FUNCTION_BLOCK J_Stop_Testing_SM
VAR_INPUT
	JST_NodeID					: BYTE; (* This Port No. addresses the CANopen Node (see System Manager) *)
	JST_Start_Testing			: BOOL; (* Send True to start the Stop Testing*)
	JST_Statusword				: WORD;	
	JST_Current_State 			: E_Statemachine_State;
END_VAR
VAR_OUTPUT
	Finished 				: BOOL;
	JST_Controlword 		: WORD;
	Mode_of_operation 		: E_Mode_of_operation	:= E_Mode_of_operation.No_mode_active;
END_VAR
VAR
	JST_Profile_Velocity_Mode 		: Profile_Velocity_Mode;
	e_Stop_Testing_State_Machine 	: (Idle,
									   Start_Drive, 
									   Check_Start_Drive_Condition,
								       Stop_Testing, 
									   Check_Stop_Drive_Condition,
									   Error_Handling) := Idle; 
									
	e_Operation_Mode : E_Mode_of_operation := E_Mode_of_operation.Profile_position_mode;
	
	e_Stop_Mode :  (Switch_On,					//schnell runterrampen -> Switched on
					Shutdown,					//Disable PS
					Disable_Voltage,			//Disable PS
					Vel_To_Zero,				//Ramp down
					Halt,						//stillstand mit dehmoment -> Weiterdrehen
					Quick_Stop,					//schnell runterrampen -> Switch on Disabled
					Fault,						//DISABLE PS
					STO1,						//Disable PS
					STO2,						//Disable PS
					END) := Switch_On;
					
	e_Stop_Type :  (Idle_Output_Stage,
				    Ramp_Down,
					Vel_Zero,
					Quick_Stop);
					
	
	JST_Profile_velocity_parameters	: ST_Velocity_parameters := (vl_target_velocity 	  := 1000,
																 vl_velocity_acceleration := 1000,
																 vl_velocity_deceleration := 1000);
	vl_target_velocity	: INT := 0;
	Target_State: E_STATEMACHINE_STATE;
	
	SDO_WRITE		: FB_SDO_WRITE;
	WriteData		: ARRAY [0..255] OF BYTE;
	
	Tolerance : INT := 30;		//Assumed that unit is RPM
	
	// Trash Variables 
	Temp : BOOL := TRUE;
	JumpNextState : BOOL := FALSE;
	
END_VAR

CASE e_Stop_Testing_State_Machine OF
	
	Idle:
		IF JST_Start_Testing THEN
			e_Stop_Testing_State_Machine := Start_Drive;
		ELSE
			e_Stop_Testing_State_Machine := Idle;
		END_IF
		
//---------------------Start Drive SM-----------------------------------
	Start_Drive:
	
		CASE e_Operation_Mode OF
			
			e_Operation_Mode.Profile_position_mode:
				// Vel = 1000 ; Acc = 1000 ; Dec = 1000, Pos = 10000000	
				IF NOT JST_Profile_Velocity_Mode.Finished THEN
					//just want to set acc and dec but not enable the drive
					JST_Profile_Velocity_Mode (NodeID := JST_NodeID,		//PVM just because the param for acc and dec are set and the same as in PPM
						   Start := TRUE,
						   Current_State := JST_Current_State,
						   Statusword := JST_Statusword,
						   Profile_velocity_parameters := JST_Profile_velocity_parameters,
						   Controlword => JST_Controlword);
					JST_Controlword := CONTROLWORD_STATE_CHANGE(JST_Current_State, E_Statemachine_State.Switch_on_disabled);
				ELSE
					WHILE Temp = TRUE DO
						PDO.Mode_of_operation 	:= E_Mode_of_operation.Profile_position_mode;		//Maybe its enought to set it once?
						PDO.Profile_velocity := JST_Profile_velocity_parameters.vl_target_velocity;
						Temp := FALSE;
					END_WHILE
					JST_Controlword := CONTROLWORD_STATE_CHANGE(JST_Current_State, E_statemachine_state.Operation_enabled);
					e_Stop_Testing_State_Machine := Check_Start_Drive_Condition;
				END_IF
								
			e_Operation_Mode.Velocity_mode:
				// Vel = 1000
				// // Start Drive, Wait for SDO written then change state
				e_Stop_Testing_State_Machine := Check_Start_Drive_Condition;
				
			e_Operation_Mode.Profile_velocity_mode:
				// Vel = 1000 ; Acc = 1000 ; Dec = 500
				// Start Drive, Wait for SDO written then change state
				e_Stop_Testing_State_Machine := Check_Start_Drive_Condition;
				
			e_Operation_Mode.Profile_torque_mode:
				// Torque = 100 pro mill
				// Start Drive, Wait for SDO written then change state
				e_Stop_Testing_State_Machine := Check_Start_Drive_Condition;
		END_CASE
		
		
//------------------Check Drive Condition SM-----------------------------
	Check_Start_Drive_Condition:
	
		CASE e_Operation_Mode OF
			
			e_Operation_Mode.Profile_position_mode:
				IF ABS(PDO.Velocity_actual_value - JST_Profile_velocity_parameters.vl_target_velocity) < Tolerance THEN
					e_Stop_Testing_State_Machine := Stop_Testing;
				ELSE
					;
				END_IF
				// Wait for desired speed 
				// true change state / false wirte msg log
			e_Operation_Mode.Velocity_mode:
				// Wait for desired speed 
				// true change state / false wirte msg log
			e_Operation_Mode.Profile_velocity_mode:
				// Check acc and dec
				// Wait for desired speed 
				// true change state / false wirte msg log
			e_Operation_Mode.Profile_torque_mode:
				// check torque
				// true change state / false wirte msg log
		END_CASE
		
//------------------Stop Testing SM--------------------------------------		
	Stop_Testing:
	
		CASE e_Operation_Mode OF
		//----------testing in Profile Position Mode---------------------
			e_Operation_Mode.Profile_position_mode:
					
				CASE e_Stop_Mode OF
					Switch_On:
						//Trigger Stopp
						e_Stop_Mode := Shutdown;
						e_Stop_Type := Idle_Output_Stage;
					Shutdown:
						//Trigger Stopp
						e_Stop_Mode := Disable_Voltage;
						e_Stop_Type := Idle_Output_Stage;
					Disable_Voltage:
						//Trigger Stopp
						e_Stop_Mode := Vel_To_Zero;
						e_Stop_Type := Idle_Output_Stage;
					Vel_To_Zero:
						//Trigger Stopp
						e_Stop_Mode := Halt;
						e_Stop_Type := Vel_Zero;
					Halt:
						//Trigger Stopp
						e_Stop_Mode := Quick_Stop;
						e_Stop_Type := Vel_Zero;
					Quick_Stop:
						//Trigger Stopp
						e_Stop_Mode := Fault;
						e_Stop_Type := Quick_Stop;
					Fault:
						//Trigger Stopp
						e_Stop_Mode := STO1;
						e_Stop_Type := Idle_Output_Stage;
					STO1:
						//Trigger Stopp
						e_Stop_Mode := STO2;
						e_Stop_Type := Idle_Output_Stage;
					STO2:
						//Trigger Stopp
						e_Stop_Mode := Switch_On;
						e_Stop_Type := Idle_Output_Stage;
						
						e_Operation_Mode := e_Operation_Mode.Velocity_mode;
				END_CASE
				e_Stop_Testing_State_Machine := Check_Stop_Drive_Condition;
				
			e_Operation_Mode.Velocity_mode:
				;
			e_Operation_Mode.Profile_velocity_mode:
				;
			e_Operation_Mode.Profile_torque_mode:
				;
		END_CASE
//---------------------Check Drive Stop------------------------------		
	Check_Stop_Drive_Condition:
		
		CASE e_Stop_Type OF
			
			Idle_Output_Stage:
				// Check for 
			Ramp_Down:
				;
			Vel_Zero:
				;
			Quick_Stop:
				;
		END_CASE
	Error_Handling:
		;
END_CASE

END_FUNCTION_BLOCK

(* stored: Version 1.1.0.1, ProductVersion 3.1.4026.11
   POU J_Stop_Testing_SM: Id {c231d705-6bba-41a2-9ea5-2d7b22a70d02}, SpecialFunc None *)
